// TIA Portal V15.1 export
// export: Created 2024-06-21T08:41:21.3804735Z, ExportSetting WithDefaults, DisplayName Totally Integrated Automation Portal, DisplayVersion V15.1 Update 5, DisplayName TIA Portal Openness, DisplayVersion V15.1 Update 5, DisplayName SINAMICS Startdrive Advanced, DisplayVersion V15.1, DisplayName G130, G150, S120, S150, SINAMICS MV, S210, DisplayVersion V15.1, DisplayName G110M, G120, G120C, G120D, G120P, DisplayVersion V15.1, DisplayName STEP 7 Professional, DisplayVersion V15.1 Update 5, DisplayName STEP 7 Safety, DisplayVersion V15.1, DisplayName WinCC Professional, DisplayVersion V15.1 Update 5, DisplayName SIMATIC Visualization Architect, DisplayVersion V15.1
FUNCTION "LAndonConfigVCG" : Void   // FC6050, FBD
TITLE = LAndonConfigVCG / LAndon-Config
{ S7_Optimized_Access := 'TRUE' }
VERSION : 0.1
// =============================================================================
// Andon Communication Configuration
// =============================================================================
// stored: AutoNumber false, IsIECCheckEnabled true, SetENOAutomatically False, UDAEnableTagReadback false
   VAR_INPUT
      C_EnableAndon : Bool;   // Enable Andon / Enable or disable AndonSystem
      C_ShopID : String;   // String Shop Id (Ex. 'GA') / Info Value VD
      C_StationCode : String;   // String Station Code ('336010ZM01' or '336010SZ01') / Info Value VD
      C_SubSystem : Int;   // Number to identify the subsystem / Identify Subsystem
      C_SubSystemMsgLenght : Int;   // Subsystem message length / Lenght of the message to be send
      C_SubSystemMsgType : Int;   // Subsystem message type / MessageType of the subsystem
      C_AlarmCFilterTime : Time;   // Alarm C filter time / Config Time Buffer Value Resend
      C_BufferValueSendFilter : Time;   // Buffer value send time / ConfigTime Resend buffer when no event occurs
      C_LocalRecvDB : DB_ANY;   // Local DB to store received data; to used by application / Local DB For Recv Data Used By The Application
      C_LocalSendDB : DB_ANY;   // Local DB for send data; to be used by application / Local DB For Send Data Used By The Application
      C_VDCommRecvDB : DB_ANY;   // VD communication system receive DB; Not to be used by application / VD communication system receive DB Not to be used by Application
      C_VDCommSendDB : DB_ANY;   // VD communication system send DB; Not to be used by application / VD communication system send DB Not to be used by Application
      C_VDCommMasterDB : DB_ANY;   // VD communication system master DB / VD Communication Master DB
   END_VAR
   VAR_IN_OUT
      IO_Config : "AndonConfigVCG";   // Config / Andon VCG Configuration
   END_VAR
BEGIN

NETWORK
TITLE = **** 1 - Inputs **** Load Config
// Load Config
      A     #C_EnableAndon;
      =     #IO_Config.AndonEnabeld;

// TRANSFER "SUBSYSTEM SETTINGS" CONFIG
      L     #C_SubSystem;
      T     #IO_Config.SubSystem;
      L     #C_SubSystemMsgType;
      T     #IO_Config.SubSystemMsgType;
      L     #C_SubSystemMsgLenght;
      T     #IO_Config.SubSystemMsgLenght;
      L     #C_LocalRecvDB;
      T     #IO_Config.LocalRecvDB;
      L     #C_LocalSendDB;
      T     #IO_Config.LocalSendDB;

// TRANSFER "VDCOM SETTINGS" CONFIG

      L     #C_VDCommRecvDB;
      T     #IO_Config.VDCommRecvDB;
      L     #C_VDCommSendDB;
      T     #IO_Config.VDCommSendDB;
      L     #C_VDCommMasterDB;
      T     #IO_Config.VDCommMasterDB;
      NOP   0;


REGION Network 2: **** 4.2 param **** Load Config
   // // TRANSFER "SHOPID" to CONFIG
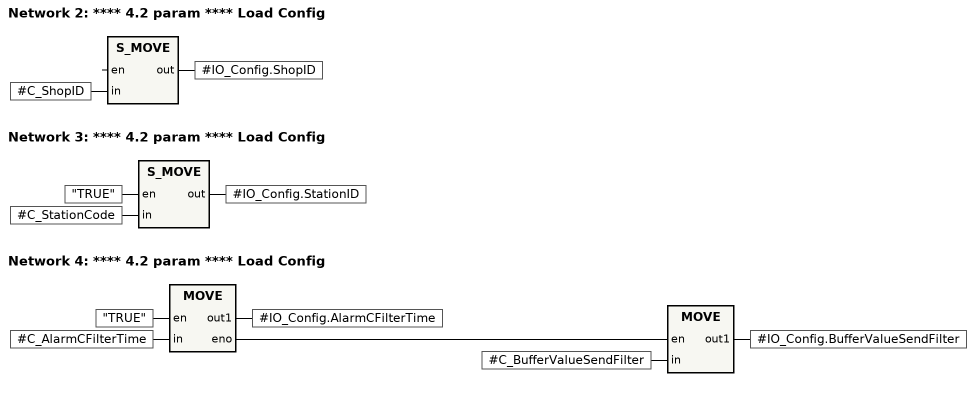
   #IO_Config.ShopID := #C_ShopID;
END_REGION

REGION Network 3: **** 4.2 param **** Load Config
   // // TRANSFER "STATIONID" to CONFIG
   IF "TRUE" THEN #IO_Config.StationID := #C_StationCode; END_IF;
END_REGION

REGION Network 4: **** 4.2 param **** Load Config
   // // TRANSFER "AlarmCFilterTime" and "BufferValueSendFilter" to CONFIG
   IF "TRUE" THEN
       #IO_Config.AlarmCFilterTime := #C_AlarmCFilterTime;
       #IO_Config.BufferValueSendFilter := #C_BufferValueSendFilter;
   END_IF;
END_REGION
END_FUNCTION
